(*
SPDX-FileCopyrightText: Â© 2026 Oleksandr Tiutyk <trofimich@gmail.com>
SPDX-License-Identifier: MIT
License: https://opensource.org/license/mit
*)

(*!
<summary>Utility program providing factory methods to construct RAW_ANALOG_VALUE unions.</summary>
<description>
Ensures that unused bytes of the 4-byte union are zero-initialized when constructing from 16-bit values.
</description>
*)

{attribute 'no_explicit_call' := 'do not call this POU directly'}
PROGRAM RawAnalogValues
VAR
	{attribute 'hide'} 
	_ClassName : STRING := __POUNAME();
END_VAR

(*!
<summary>Gets the class name of the program.</summary>
*)
{attribute 'monitoring' := 'call'}
PROPERTY ClassName : REFERENCE TO STRING
GET
ClassName REF= _ClassName;
END_GET
END_PROPERTY

(*!
<summary>Creates a RAW_ANALOG_VALUE union from a 16-bit signed integer.</summary>
<description>Zeroes upper bytes of the 4-byte union before assigning the 16-bit value.</description>
<param name="value">16-bit signed integer value.</param>
*)
METHOD FromInt16 : RAW_ANALOG_VALUE
VAR_INPUT
	value : INT;
END_VAR
FromInt16.Int32 := 0;
FromInt16.Int16 := value;
END_METHOD

(*!
<summary>Creates a RAW_ANALOG_VALUE union from a 32-bit signed integer.</summary>
<param name="value">32-bit signed integer value.</param>
*)
METHOD FromInt32 : RAW_ANALOG_VALUE
VAR_INPUT
	value : DINT;
END_VAR
FromInt32.Int32 := value;
END_METHOD

(*!
<summary>Creates a RAW_ANALOG_VALUE union from a 32-bit single-precision float.</summary>
<param name="value">32-bit float value.</param>
*)
METHOD FromReal32 : RAW_ANALOG_VALUE
VAR_INPUT
	value : REAL;
END_VAR
FromReal32.Real32 := value;
END_METHOD

(*!
<summary>Gets the namespace name of the program.</summary>
*)
{attribute 'monitoring' := 'call'}
PROPERTY NamespaceName : REFERENCE TO STRING
GET
NamespaceName REF= CurrentNamespace.Name;
END_GET
END_PROPERTY

END_PROGRAM

(* stored: Version 1.1.0.1
   POU RawAnalogValues: Id {2cbcd7e2-bc1d-44e8-a9a9-a10af65b8b2d}, SpecialFunc None
   Property ClassName: Id {b34f30ae-eca8-45b9-88f9-c1b0b9ee84e8}
   Get Get: Id {d4a4c5c6-9279-4e80-bcb3-1ff73bc61b4c}
   Method FromInt16: Id {32647063-a064-4305-908f-8b4e3f2aa8c3}
   Method FromInt32: Id {ab5fb223-7868-464d-b37e-4693aa2f3aef}
   Method FromReal32: Id {1eb223f2-6255-44c9-83fa-26b2a8cc65a0}
   Property NamespaceName: Id {b5f61307-0199-4210-84f3-a3306f1e01dc}
   Get Get: Id {f506b0a8-306c-4d6b-ac5a-29b295f521d1} *)
